// TwinCAT 3 PLC project CX2043_0175
// ProgramVersion: 3.1.4024.0
// libraries:
//   Tc2_Standard, * (Beckhoff Automation GmbH)
//   Tc2_System, * (Beckhoff Automation GmbH)
//   Tc3_Database, * (Beckhoff Automation GmbH)
//   Tc3_EventLogger, * (Beckhoff Automation GmbH)
//   Tc3_Module, * (Beckhoff Automation GmbH)
// project tree:
//   DUTs/ ST_ErrorEntry.TcDUT, ST_SearchData.TcDUT
//   GVLs/ Alarm.TcGVL, GVL_CONSTANT.TcGVL, HMI.TcGVL, IOs.TcGVL
//   Logger/ FB_ErrorLogger.TcPOU
//   / PlcTask.TcTTO
//   POUs/Alarm/ FB_Alarm.TcPOU
//   POUs/DigitalInput/ FB_DidigtalInputSensor.TcPOU
//   POUs/LightTower/ BuzzerType.TcDUT, LightTower.TcPOU, LightType.TcDUT
//   POUs/Loadcell/ FB_Loadcell.TcPOU
//   POUs/ MAIN.TcPOU
//   POUs/Slider/ FB_Slider.TcPOU
// real-time tasks:
//   TASK PlcTask: cycle T#10ms, priority 20, ADS port 350
// I/O:
//   DEVICE Device 1 (EtherCAT) (disabled), AmsNetId 192.168.68.53.3.1
//     Term 9 (EK1200) [EK1200-5000 EtherCAT Power supply (2A E-Bus)]
//       #Slot 1 (EL1819) [EL1819 16Ch. Dig. Input 24V, 10µs]
//       #Slot 2 (EL1819) [EL1819 16Ch. Dig. Input 24V, 10µs]
//       #Slot 3 (EL1819) [EL1819 16Ch. Dig. Input 24V, 10µs]
//       #Slot 4 (EL2809) [EL2809 16Ch. Dig. Output 24V, 0.5A]
//       #Slot 5 (EL9410) [EL9410 E-Bus Power Supplier  (Diagnostics)]
//       #Slot 6 (EL2809) [EL2809 16Ch. Dig. Output 24V, 0.5A]
//       #Slot 7 (EK1122) [EK1122 2 port EtherCAT junction]
//       #Slot 8 (EL3124) [EL3124 4Ch. Ana. Input 4-20mA Diff.]
//       #Slot 9 (EL9410) [EL9410 E-Bus Power Supplier  (Diagnostics)]
//       #Slot 10 (EL9011) [EL9011 End Terminal]

CONFIGURATION CX2043_0175
    RESOURCE PLC ON TwinCAT3
        TASK PlcTask(INTERVAL := T#10ms, PRIORITY := 20);
        PROGRAM MAIN WITH PlcTask : MAIN;
    END_RESOURCE
END_CONFIGURATION

// ---- DUTs/ST_ErrorEntry.TcDUT
TYPE ST_ErrorEntry :
STRUCT
	tTimestamp : DT;
	nErrCode : UDINT;
	sSeverity : STRING(10);	
	sMsg : T_MaxString;
END_STRUCT
END_TYPE

// ---- DUTs/ST_SearchData.TcDUT
TYPE ST_SearchData :
STRUCT
	dtStartTimestamp : DT;
	dtEndTimestamp : DT;
END_STRUCT
END_TYPE

// ---- POUs/LightTower/BuzzerType.TcDUT
{attribute 'qualified_only'}
{attribute 'strict'}
TYPE BuzzerType :
(
	ONCE := 0,
	CYCLE,
	OFF
);
END_TYPE

// ---- POUs/LightTower/LightType.TcDUT
{attribute 'qualified_only'}
{attribute 'strict'}
TYPE LightType :
(
	ON := 0,
	FLASH,
	OFF
);
END_TYPE

// ---- GVLs/Alarm.TcGVL
{attribute 'qualified_only'}
VAR_GLOBAL CONSTANT
	//Setting constants alarm range
	
	//Loadcell sensor S13
	minAlarm_loadcell : UINT := 0;
	maxAlarm_loadcell : UINT := 240; //[TBD]
	
	//Material tray sensor S24
	maxAlarm_finishTray : UINT := 80; //[TBD]
	
	
END_VAR

VAR_GLOBAL
	//General alarm
	
	//Material tray alarm-----------------------------------------------------
	
	//Material tray installation sensor
	materialTray_notInstalled : BOOL ; //sensor S0
	materialTray_empty 		  : BOOL ; //sensor S1 & S2
	
	//Cylinder C1 sensor
	cylinderC1_retractTimeout : BOOL ; //Sensor S3
	cylinderC1_extractTimeout : BOOL ; //Sensor S4
	
	//Cylinder C2 sensor
	cylinderC2_retractTimeout : BOOL ; //Sensor S6
	cylinderC2_extractTimeout : BOOL ; //Sensor S5
	
	//Cylinder C3 sensor
	cylinderC3_retractTimeout : BOOL ; //Sensor S8
	cylinderC3_extractTimeout : BOOL ; //Sensor S7
	
	//Material counting S9 sensor
	materialCover_countingSensor : BOOL ; //Sensor S9
	
	
	
	//Feeder alarm -----------------------------------------------------------
	
	//Material in position of roller M1
	feederSensor_rollerM1 : BOOL ; //Sensor S12
	
	//Roller M1
	rollerM1_error : BOOL ; //Error from roller M1 controller
	
	//Cylinder C5
	cylinderC5_extractTimeout : BOOL ; //Sensor S14
	cylinderC5_retractTimeout : BOOL ; //Sensor S15
	
	
	
	//Stripping alarm--------------------------------------------------------
	
	//Cylinder C6
	cylinderC6_extractTimeout : BOOL ; //Sensor S16
	cylinderC6_retractTimeout : BOOL ; //Sensor S17
	
	//Material in position of roller M2
	feederSensor_RollerM2 : BOOL ; //Sensor S20
	
	//Roller M2
	rollerM2_error : BOOL ; //Error from roller M2 controller
	
	//CO2 lazer error
	lazerCO2_error : BOOL ; //Error from CO2 lazer
	
	//UV lazer error
	lazerUV_error  : BOOL ; //Error from UV lazer
	
	
	
	//Grinding alarm--------------------------------------------------------
	
	//Roller M3
	rollerM3_error : BOOL ; //Error from roller M3 controller
	
	//Cylinder C7
	cylinderC7_extractTimeout : BOOL ; //Sensor S18
	cylinderC7_retractTimeout : BOOL ; //Sensor S19
	
	//Cylinder C8
	cylinderC8_extractTimeout : BOOL ; //Sensor S25
	cylinderC8_retractTimeout : BOOL ; //Sensor S26
	
	//Gripper roller M4
	grindingPosition_timeout : BOOL ; //Sensor S21
	//Gripper position
	gripperPosition_timeout  : BOOL ; //Sensor S22
	//Home position
	homePosition_timeout     : BOOL ; //Sensor S23
	//Roller M4
	rollerM4_error           : BOOL ; //Error from roller M4 controller
	
	//Slider error
	//Idle position
	idleSLIR_timeout     : BOOL ; //Sensor S27 at waiting position
	//Grinding position
	grindingSLIR_timeout : BOOL ; //Sensor S10 at grinding & gripping position
	//Home position
	homeSLIR_timeout     : BOOL ; //Sensor S11 at home position
	//Slider
	SLIR_error           : BOOL ; //Slider error from controller
	
	//Finish good tray
	finishGoodTray_timeout : BOOL ; //Sensor S24 - analog error when timeout (after TBD cycle)
	
	
	
	//Frame alarm-----------------------------------------------------------
	
	//EMS button
	buttonEMS_pressed : BOOL ; //EMS button is active status
	
	//Left door interlock
	leftDoorOpening_timeout : BOOL ; //Left door opening timeout
	leftDoorLock_timeout    : BOOL ; //Left door lock timeout
	
	//Right door interlock
	rightDoorOpening_timeout : BOOL ; //Right door opening timeout
	rightDoorLock_timeout    : BOOL ; //Right door lock timeout
	
	//[TBD]High air-pressure level
	//highAirPressure_alarm : BOOL ; //Current air-pressure over operation range
	//[TBD]Low air-pressure level
	//lowAirPressure_alarm  : BOOL ; //Current air-pressure lower operation range
	
	//Safety relay
	safetyRelay_active : BOOL ; //Safety relay active
	
	
END_VAR

// ---- GVLs/GVL_CONSTANT.TcGVL
{attribute 'qualified_only'}
VAR_GLOBAL CONSTANT
	
END_VAR

// ---- GVLs/HMI.TcGVL
{attribute 'qualified_only'}
VAR_GLOBAL

{region Buttons}
	//Operational Controls-------
	//Run Button
	runButton : BOOL;
	//Stop Button
	stopButton : BOOL;
	//Reset Button
	resetButton : BOOL;
	//Calibration Mode Button - Only display with maintenance authentication
	calibButton : BOOL;
	//Auto/Manual Mode
	autoManualMode : BOOL;
{endregion}
	 
{region System Status}
	//Overall system status--------------
	//System ready
	sysReady : BOOL;
	//System error
	sysError : BOOL;
	//System running
	sysRunning : BOOL;
{endregion}

END_VAR

// ---- GVLs/IOs.TcGVL
{attribute 'qualified_only'}
VAR_GLOBAL
///Inputs ================================================================================================================================================================
	
	///Digital ********************************************************
	
	//Operation Control Buttons
	//Start Push Button
	startButton AT %I* : BOOL;
	
	//Stop Push Button
	stopButton AT %I* : BOOL;
	
	//Reset Push Button
	resetButton AT %I* : BOOL;
	
	//E-Stop Status : True if OK, False is E-Stop is enabled
	eStop AT %I* : BOOL;
	
	
	// Feeder and Stripping Section -----------------------------------
	
	//Material tray installation sensor
	S0 AT %I* : BOOL;
	
	//Counting material cover sensor
	S9 AT %I* : BOOL;
	
	//Material in position roller M1 sensor
	S12 AT %I* : BOOL;
	
	// Materials in tray sensor
	S1 AT %I* : BOOL;
	S2 AT %I* : BOOL;
	
	// Cylinder C1 : Position sensor
	// Cylinder C1 retract
	S4 AT %I* : BOOL;
	// Cylinder C1 extract
	S3 AT %I* : BOOL;
	
	// Cylinder C2 and C3 : Position sensor
	// Cylinder C2 and C3 extract
	S5 AT %I* : BOOL;
	S7 AT %I* : BOOL;
	// Cylinder C2 and C3 retract
	S6 AT %I* : BOOL;
	S8 AT %I* : BOOL;

	// Cylinder C5 : Position sensor
	// Cylinder C5 extract
	S14 AT %I* : BOOL;
	// Cylinder C5 retract
	S15 AT %I* : BOOL;
	
	// Cylinder C6 : Position sensor
	// Cylinder C6 retract
	S16 AT %I* : BOOL;
	// Cylinder C6 extract
	S17 AT %I* : BOOL;
	
	
	// Grinding Section -----------------------------------------------

	//Slider position sensor
	//Grinding position sensor
	S10 AT %I* : BOOL;
	//Stripping position sensor
	S11 AT %I* : BOOL;
	
	// Cylinder C7 retract
	S18 AT %I* : BOOL;
	// Cylinder C7 extract
	S19 AT %I* : BOOL;
	
	//Material in position roller M3
	S20 AT %I* : BOOL;

	//Swing arm position sensors
	//Home position sensor
	S21 AT %I* : BOOL;
	
	//Grinding position sensor
	S22 AT %I* : BOOL;
	
	//Extract finish good position sensor
	S23 AT %I* : BOOL;

	//System Input----------------------------------------------------
	
	//Left Door Interlock
	//Door interlock left: left door open (open = 1; close = 0)
	LDO AT %I* : BOOL;
	//Door interlock left: left door locked (unlock = 1; locked = 0)
	LDL AT %I* : BOOL;
	
	//Right Door Interlock
	//Door interlock right: right door open (open = 1; close = 0)
	RDO AT %I* : BOOL;
	//Door interlock right: right door locked (unlock = 1; locked = 0)
	RDL AT %I* : BOOL;
	
	//Lazer Control Input
	//UV Lazer running
	UV_Running AT %I* : BOOL;
	//UV Lazer finish
	UV_Finish AT %I* : BOOL;
	//UV Lazer error
	UV_Error AT %I* : BOOL;
	
	//CO2 Lazer running
	CO2_Running AT %I* : BOOL;
	//CO2 Lazer finish
	CO2_Finish AT %I* : BOOL;
	//CO2 Lazer error
	CO2_Error AT %I* : BOOL;

	//Electrical cabinet limit switch
	//AC Cabinet limit switch
	AC_Limit AT %I* : BOOL;
	
	//DC Cabinet limit switch
	DC_Limit AT %I* : BOOL;
	
	//Air pressure sensor
	highLevelPressure  AT %I* : BOOL;
	howLevelPressure   AT %I* : BOOL;
	
	//Safety relay status
	safetyRelay_Status AT %I* : BOOL;
	
	
	///Analog ********************************************************
	//EL3124 output values:
	// 4 mA -  0
	// 12 mA - 16383
	// 20 mA - 32767
	S13_Loadcell AT %I* : INT; //grinding loadcell
	S24_Analog 	 AT %I* : INT; //finish good material tray
	
	//Grinding loadcell sensor
	S13 AT %I* : INT;
	
	// Finish good tray sensor
	S24 AT %I* : INT;


///Outputs ===============================================================================================================================================================
	
	///Digital ********************************************************
	
	//1. Lazer control
	ena_UVLazer       AT %Q* : BOOL;
	ena_CO2Lazer      AT %Q* : BOOL;
	
	//2. Cylinder control
	cylinderC1_Extract   AT %Q* : BOOL;
	cylinderC1_Retract   AT %Q* : BOOL;
	cylinderC2n3_Extract AT %Q* : BOOL;
	cylinderC2n3_Retract AT %Q* : BOOL;
	cylinderC5_Extract   AT %Q* : BOOL;
	cylinderC5_Retract   AT %Q* : BOOL;
	cylinderC6_Extract   AT %Q* : BOOL;
	cylinderC6_Retract   AT %Q* : BOOL;
	cylinderC7_Extract   AT %Q* : BOOL;
	cylinderC7_Retract   AT %Q* : BOOL;
	cylinderC8_Extract   AT %Q* : BOOL;
	cylinderC8_Retract   AT %Q* : BOOL;
	
	//3. Fume fan control
	fumeFan  AT %Q* : BOOL;
	
	//4. Illuminated control buttons
	illuminatedStart  AT %Q* : BOOL;
	illuminatedStop   AT %Q* : BOOL;
	
	///Safety Control Digital Output

	//1. Light Tower
    lightTowerRed     AT %Q* : BOOL;
    lightTowerYellow  AT %Q* : BOOL;
    lightTowerGreen	  AT %Q* : BOOL;
	lightTowerBuzzer  AT %Q* : BOOL;
	
	//2. Safety relay activate
	safetyRelayActive  AT %Q* : BOOL;
	
	//3. Door interlock
	lock_LeftDoor   AT %Q* : BOOL;
	lock_RightDoor  AT %Q* : BOOL;
	
	//4. 
	
END_VAR

// ---- POUs/MAIN.TcPOU
PROGRAM MAIN

VAR
	//S1 : digitalInputSensor;
	temp_S : BOOL;
	digitalInputSensor: INT;
	materialTrayInstallationSensor: INT;
END_VAR

//S1();
//S1(on := IOs.S1, inTime := T#50MS, digitalFiltered => temp_S);

//digitalInputSensor.materialTrayInstallationSensor(temp_S);

END_PROGRAM

// ---- Logger/FB_ErrorLogger.TcPOU
FUNCTION_BLOCK PUBLIC FB_ErrorLogger
VAR_INPUT
	
END_VAR
VAR_OUTPUT
	
END_VAR
VAR
	
END_VAR

END_FUNCTION_BLOCK

// ---- POUs/Alarm/FB_Alarm.TcPOU
FUNCTION_BLOCK FB_Alarm
VAR_INPUT
	
	//Error/Warning from devices
	safetyRelay : BOOL;
	sensorTimeout : BOOL;
	actuatorWarning : BOOL;
	controllerWarning : BOOL;
	
END_VAR

VAR_OUTPUT
	//Enable system when no error and disable system when error
	sysEnable : BOOL;
	sysHome : BOOL;
	
END_VAR

VAR
	//Operation status to devices
	stopCase : BOOL;
	resetCase : BOOL;
	runCase : BOOL;
	homing : BOOL;
	
END_VAR

//When safety relay active -> stop system and reset system when back to run status.
IF safetyRelay THEN
	stopCase := TRUE;
	sysEnable := FALSE;
	homing := TRUE;
ELSIF homing AND NOT safetyRelay THEN
	sysHome := TRUE;
	resetCase := TRUE;
	sysEnable := TRUE;
	homing := FALSE;
ELSIF NOT safetyRelay AND NOT homing THEN
	sysHome := FALSE;
END_IF

//When sensor timeout -> stop system and continue to run when back to run status.
IF sensorTimeout OR actuatorWarning OR controllerWarning THEN
	sysEnable := FALSE;
	stopCase := TRUE;
ELSE sysEnable := TRUE; runCase := TRUE;
END_IF

METHOD cylinders : BOOL
VAR_INPUT
END_VAR
END_METHOD

METHOD detectSensors : BOOL
VAR_INPUT
END_VAR
END_METHOD

METHOD doorInterlock : BOOL
VAR_INPUT
END_VAR
END_METHOD

METHOD safetyRelay : BOOL
VAR_INPUT
END_VAR
END_METHOD

METHOD slider : BOOL
VAR_INPUT
END_VAR
END_METHOD

END_FUNCTION_BLOCK

// ---- POUs/DigitalInput/FB_DidigtalInputSensor.TcPOU
FUNCTION_BLOCK FB_DigitalInputSensor
VAR_INPUT
	on : BOOL;
	inTime : TIME;
	
END_VAR

VAR_OUTPUT
	digitalFiltered : BOOL;
END_VAR
VAR
	tOnGetTime : TON;
END_VAR

tOnGetTime(PT := inTime);
IF on THEN
	tOnGetTime.IN := TRUE;
	IF tOnGetTime.Q THEN
		digitalFiltered := TRUE;
	ELSE digitalFiltered := FALSE;
	END_IF
ELSE tOnGetTime.IN := FALSE;
END_IF

END_FUNCTION_BLOCK

// ---- POUs/LightTower/LightTower.TcPOU
FUNCTION_BLOCK LightTower
VAR_INPUT
	buzzerMute : BOOL := FALSE;
	cycle_light_time 	: TIME 		:= T#1S;
END_VAR
VAR_OUTPUT
END_VAR
VAR
	m_red   		: BOOL		:= FALSE;
	m_yellow 		: BOOL		:= FALSE;
	m_green 		: BOOL		:= FALSE;
	m_buzzer  		: BOOL		:= FALSE;
	
	flash_light 	: BOOL := TRUE;
	flash_buzzer 	: BOOL := TRUE;
	
	timer_light 	: TON;

	timer_cyclebuzzer	: TON;
	cycle_buzzer_time 	: TIME 		:= T#3S;
	
	timer_oncebuzzer	: TON;
	once_buzzer_time 	: TIME 		:= T#0.5S;
	
	enableCycleBuzzer 	: BOOL;
	enableOnceBuzzer 	: BOOL;
END_VAR

// flash light
timer_light(IN := TRUE, PT := cycle_light_time);
IF timer_light.Q THEN
	flash_light := NOT flash_light;
	timer_light(IN := FALSE);
END_IF

// cycle buzzer 
IF enableCycleBuzzer THEN
	timer_cyclebuzzer(IN := TRUE, PT := cycle_buzzer_time);
	IF timer_cyclebuzzer.Q THEN
		flash_buzzer := NOT flash_buzzer;
		timer_cyclebuzzer(IN := FALSE);
	END_IF
ELSE
	flash_buzzer := TRUE;
	timer_cyclebuzzer(IN := FALSE);
END_IF

//once buzzer
IF enableOnceBuzzer THEN
	timer_oncebuzzer(IN := TRUE, PT := once_buzzer_time);
	IF timer_oncebuzzer.Q THEN
		runBuzzer(BuzzerType.OFF,once_buzzer_time);
		enableOnceBuzzer := FALSE;
		timer_oncebuzzer(IN := FALSE);
	END_IF
END_IF

IF buzzerMute THEN
	m_buzzer := FALSE;
END_IF
/////////////////
onCycle();

METHOD PRIVATE onCycle : BOOL
VAR_INPUT
END_VAR
IOs.lightTowerRed   	:= m_red;
IOs.lightTowerYellow := m_yellow;
IOs.lightTowerGreen 	:= m_green;
IOs.lightTowerBuzzer := m_buzzer;
END_METHOD

METHOD PUBLIC runBuzzer : BOOL
VAR_INPUT
	//enable  : BOOL;
	event : BuzzerType;
	timeBuzzer : TIME;
END_VAR
cycle_buzzer_time := timeBuzzer;
IF NOT buzzerMute THEN
	IF event = BuzzerType.CYCLE THEN
		m_buzzer := flash_buzzer;
		enableCycleBuzzer := TRUE;
		enableOnceBuzzer := FALSE;
	ELSIF event = BuzzerType.ONCE THEN
		m_buzzer := TRUE;
		enableCycleBuzzer := FALSE;
		enableOnceBuzzer := TRUE;
	ELSIF event = BuzzerType.OFF THEN
		enableCycleBuzzer := FALSE;
		enableOnceBuzzer := FALSE;
		m_buzzer := FALSE;
	END_IF
END_IF
END_METHOD

METHOD PUBLIC runGreenLight : BOOL
VAR_INPUT
	enable  : BOOL;
	event 	: LightType := LightType.ON;
END_VAR
IF event = LightType.FLASH AND enable THEN
	m_green := flash_light;//flash
ELSE
	m_green := enable;
END_IF
END_METHOD

METHOD PUBLIC runRedLight : BOOL
VAR_INPUT
	enable  : BOOL;
	event 	: LightType := LightType.ON;
END_VAR
IF event = LightType.FLASH AND enable THEN
	m_red := flash_light;//flash
ELSE
	m_red := enable;
END_IF
END_METHOD

METHOD PUBLIC runYellowLight : BOOL
VAR_INPUT
	enable  : BOOL;
	event 	: LightType := LightType.ON;
END_VAR
IF event = LightType.FLASH AND enable THEN
	m_yellow := flash_light;//flash;
ELSE
	m_yellow := enable;
END_IF
END_METHOD

END_FUNCTION_BLOCK

// ---- POUs/Loadcell/FB_Loadcell.TcPOU
FUNCTION_BLOCK FB_Loadcell
VAR_INPUT
    analogInput : INT;       
    timeSpan : TIME := T#50MS; //Sample time
END_VAR

VAR_OUTPUT
    filteredOutput : REAL; 
END_VAR

VAR
    buffer : ARRAY[1..100] OF INT; //Array to save input value to buffer memory
    bufferIndex : INT := 1;        //Current index to specify next value for register
    lastUpdateTime : TIME;
    currentTime : TIME;
    sum : LREAL := 0;              // Sum of input value
    count : INT := 0;
	sysTimeGet: TIME;
END_VAR

IF NOT (sysTimeGet(currentTime) = 0) THEN
    // Check the passed time from last update
    IF (currentTime - lastUpdateTime) >= timeSpan THEN
        // Save new value to buffer memory
        sum := sum - buffer[bufferIndex]; //Remove old value from buffer memory
        buffer[bufferIndex] := analogInput; // Regist new value to buffer memory
        sum := sum + analogInput; // + new value to buffer memory

        // update buffer index
        bufferIndex := bufferIndex + 1;
        IF bufferIndex > 100 THEN
            bufferIndex := 1; // return to first value of buffer memory
        END_IF;

        //update number of value in buffer memory
        IF count < 100 THEN
            count := Count + 1;
        END_IF;

        
        filteredOutput := REAL(sum) / REAL(count);

        // update time
        lastUpdateTime := currentTime;
    END_IF;
END_IF;

END_FUNCTION_BLOCK

// ---- POUs/Slider/FB_Slider.TcPOU
FUNCTION_BLOCK FB_Slider
VAR_INPUT
END_VAR
VAR_OUTPUT
END_VAR
VAR
END_VAR

END_FUNCTION_BLOCK
